FUNCTION_BLOCK RequestResolver
  (* Standard: 61499-2 *)
  (* Version 0.1, 2014-00-16, Canto-Air, CANTO-AIR-PC *)
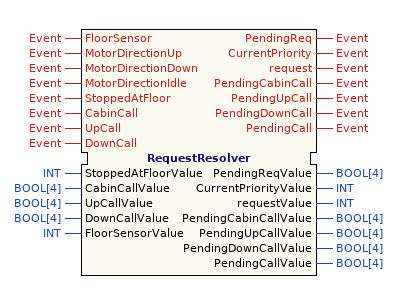
  EVENT_INPUT
    FloorSensor;
    MotorDirectionUp;
    MotorDirectionDown;
    MotorDirectionIdle;
    StoppedAtFloor;
    CabinCall;
    UpCall;
    DownCall;
  END_EVENT
  EVENT_OUTPUT
    PendingReq;
    CurrentPriority;
    request;
    PendingCabinCall;
    PendingUpCall;
    PendingDownCall;
    PendingCall;
  END_EVENT
  VAR_INPUT
    StoppedAtFloorValue : INT;
    CabinCallValue : ARRAY [0..3] OF BOOL;
    UpCallValue : ARRAY [0..3] OF BOOL;
    DownCallValue : ARRAY [0..3] OF BOOL;
    FloorSensorValue : INT;
  END_VAR
  VAR_OUTPUT
    PendingReqValue : ARRAY [0..3] OF BOOL;
    CurrentPriorityValue : INT;
    requestValue : INT;
    PendingCabinCallValue : ARRAY [0..3] OF BOOL;
    PendingUpCallValue : ARRAY [0..3] OF BOOL;
    PendingDownCallValue : ARRAY [0..3] OF BOOL;
    PendingCallValue : ARRAY [0..3] OF BOOL;
  END_VAR
  FBS
    PendingRequestGenerator : PendingRequestGenerator;
    HighestRequestProducer : HighestRequestProducer;
    RequestConsumer : RequestConsumer;
  END_FBS
  EVENT_CONNECTIONS
    FloorSensor TO HighestRequestProducer.FloorSensor;
    MotorDirectionUp TO HighestRequestProducer.MotorDirectionUp;
    MotorDirectionUp TO PendingRequestGenerator.MotorDirectionUp;
    MotorDirectionDown TO HighestRequestProducer.MotorDirectionDown;
    MotorDirectionDown TO PendingRequestGenerator.MotorDirectionDown;
    MotorDirectionIdle TO HighestRequestProducer.MotorDirectionIdle;
    StoppedAtFloor TO RequestConsumer.StoppedAtFloor;
    StoppedAtFloor TO PendingRequestGenerator.StoppedAtFloor;
    CabinCall TO PendingRequestGenerator.CabinCall;
    UpCall TO PendingRequestGenerator.UpCall;
    DownCall TO PendingRequestGenerator.DownCall;
    PendingRequestGenerator.PendingReq TO PendingReq;
    HighestRequestProducer.CurrentPriority TO CurrentPriority;
    RequestConsumer.request TO request;
    PendingRequestGenerator.PendingCabinCall TO PendingCabinCall;
    PendingRequestGenerator.PendingUpCall TO PendingUpCall;
    PendingRequestGenerator.PendingDownCall TO PendingDownCall;
    PendingRequestGenerator.PendingCall TO PendingCall;
    PendingRequestGenerator.PendingReq TO HighestRequestProducer.PendingReq;
    HighestRequestProducer.CurrentPriority TO RequestConsumer.CurrentPriority;
  END_CONNECTIONS
  DATA_CONNECTIONS
    FloorSensorValue TO HighestRequestProducer.FloorSensorValue;
    StoppedAtFloorValue TO RequestConsumer.StoppedAtFloorValue;
    StoppedAtFloorValue TO PendingRequestGenerator.StoppedAtFloorValue;
    CabinCallValue TO PendingRequestGenerator.CabinCallValue;
    UpCallValue TO PendingRequestGenerator.UpCallValue;
    DownCallValue TO PendingRequestGenerator.DownCallValue;
    PendingRequestGenerator.PendingReqValue TO PendingReqValue;
    HighestRequestProducer.CurrentPriorityValue TO CurrentPriorityValue;
    RequestConsumer.requestValue TO requestValue;
    PendingRequestGenerator.PendingCabinCallValue TO PendingCabinCallValue;
    PendingRequestGenerator.PendingUpCallValue TO PendingUpCallValue;
    PendingRequestGenerator.PendingDownCallValue TO PendingDownCallValue;
    PendingRequestGenerator.PendingCallValue TO PendingCallValue;
    PendingRequestGenerator.PendingReqValue TO HighestRequestProducer.PendingReqValue;
    HighestRequestProducer.CurrentPriorityValue TO RequestConsumer.CurrentPriorityValue;
  END_CONNECTIONS
END_FUNCTION_BLOCK
